// TIA Portal project "Software Day8" (V15)

(* hardware
DEVICE "S7-1200 station_1"  S7-1200 Station
   slot 0: "Rack_0"  S7-1200 Rack  Rack  V1.0
   slot 1: "PLC_1"  CPU 1215C AC/DC/Rly  6ES7 215-1BG40-0XB0  V4.0
*)

// ===== PLC "PLC_1"  CPU 1215C AC/DC/Rly =====

VAR_GLOBAL   // PLC tag table "Default tag table"
   "Tag_1" AT %MD100 : Real;
END_VAR

VAR_GLOBAL   // PLC tag table "VARI"
   "Start" AT %M0.0 : Bool;
   "Pump_A" AT %Q0.0 : Bool;
   "Pump_B" AT %Q0.1 : Bool;
   "Pump_C" AT %Q0.2 : Bool;
   "Mixer Motor" AT %Q0.3 : Bool;
   "Drain Valve" AT %Q0.4 : Bool;
   "Halt" AT %M0.1 : Bool;
   "Empty Sensor" AT %Q0.5 : Bool;
   "Timer 4 CV" AT %MD2 : Time;
   "Stop" AT %M0.2 : Bool;
   "Reset" AT %M0.3 : Bool;
   "Pump A Value" AT %MW64 : Word;
   "Pump B Value" AT %MW66 : Word;
   "Pump C Value" AT %MW68 : Word;
   "Pump A Norm" AT %MD6 : Real;
   "Pump B Norm" AT %MD10 : Real;
   "Pump C Norm" AT %MD14 : Real;
   "Pump A Scaled" AT %MD18 : Real;
   "Pump B Scaled" AT %MD22 : Real;
   "Pump C Scaled" AT %MD26 : Real;
   "Pump A Flow" AT %MD30 : Real;
   "Pump B Flow" AT %MD34 : Real;
   "Pump C Flow" AT %MD38 : Real;
   "Current Level" AT %MD42 : Real;
   "Previous Level" AT %MD46 : Real;
   "Actual Flow Rate" AT %MD50 : Real;
   "ETT" AT %MD54 : DInt;
   "Elapsed Time" AT %MD58 : Real;
   "Expected Flow Rate" AT %MD72 : Real;
   "Flow Rate Diff" AT %MD76 : Real;
   "Flow Rate Mismatch" AT %Q0.7 : Bool;
   "High Level Sensor" AT %Q1.0 : Bool;
   "RED ALARM" AT %Q1.1 : Bool;
   "Current Cycle State" AT %Q1.2 : Bool;
   "Current Step" AT %MW10 : Int;
   "Start Next Cycle" AT %M0.4 : Bool;
   "Flow Rate Difference" AT %MD80 : Real;
END_VAR

// folder: System blocks/Program resources

DATA_BLOCK "IEC_Timer_0_DB"   // DB1
{ S7_Optimized_Access := 'TRUE' }
AUTHOR : Simatic
FAMILY : IEC
NAME : IEC_TMR
VERSION : 1.0
// stored: InstanceOfName IEC_TIMER
"IEC_TIMER"
BEGIN
END_DATA_BLOCK

DATA_BLOCK "IEC_Counter_0_DB"   // DB4
{ S7_Optimized_Access := 'TRUE' }
AUTHOR : Simatic
FAMILY : IEC
NAME : CNTR
VERSION : 1.0
// stored: InstanceOfName IEC_COUNTER
"IEC_COUNTER"
BEGIN
END_DATA_BLOCK

DATA_BLOCK "Timer 1"   // DB6
{ S7_Optimized_Access := 'TRUE' }
AUTHOR : Simatic
FAMILY : IEC
NAME : IEC_TMR
VERSION : 1.0
// stored: InstanceOfName IEC_TIMER
"IEC_TIMER"
BEGIN
END_DATA_BLOCK

DATA_BLOCK "Timer 2"   // DB7
{ S7_Optimized_Access := 'TRUE' }
AUTHOR : Simatic
FAMILY : IEC
NAME : IEC_TMR
VERSION : 1.0
// stored: InstanceOfName IEC_TIMER
"IEC_TIMER"
BEGIN
END_DATA_BLOCK

DATA_BLOCK "Timer 3"   // DB8
{ S7_Optimized_Access := 'TRUE' }
AUTHOR : Simatic
FAMILY : IEC
NAME : IEC_TMR
VERSION : 1.0
// stored: InstanceOfName IEC_TIMER
"IEC_TIMER"
BEGIN
END_DATA_BLOCK

DATA_BLOCK "Timer 4"   // DB9
{ S7_Optimized_Access := 'TRUE' }
AUTHOR : Simatic
FAMILY : IEC
NAME : IEC_TMR
VERSION : 1.0
// stored: InstanceOfName IEC_TIMER
"IEC_TIMER"
BEGIN
END_DATA_BLOCK

// folder: (top level)

ORGANIZATION_BLOCK "Main"   // OB1, LAD, ProgramCycle
TITLE = "Main Program Sweep (Cycle)"
{ S7_Optimized_Access := 'TRUE' }
VERSION : 0.1
// The "Smart" Chemical Dosing Tank (Difficulty: Advanced - Capstone)
// 
// Scenario:
// A tank must mix 3 liquids (A, B, and C) according to a recipe. The PLC controls the pumps using timers. However, the pumps wear out, so the PLC auto-adjusts the timer presets based on a real-time flow rate derived from level sensors.
// 
// 1. Sequential Filling (Timers):
// High_Level (At 90% full).
// Outputs: Pump_A, Pump_B, Pump_C, Mixer_Motor, Drain_Valve.
// Turn on Pump_A for Preset_A seconds. Stop it. Turn on Pump_B for Preset_B seconds. Stop it. Turn on Pump_C for Preset_C seconds. Stop it. Then run the Mixer Motor for 10 seconds. Finally, open the Drain_Valve until the Empty_Sensor triggers. This is a continuous batch cycle.
// 
// 2. Batch Counter (Counters): Use a CTU to count how many complete batches (drain cycles) are finished.
// 
// 3. Adaptive Flow Correction (Math & Comparators):
// Premise: Pump_A is supposed to deliver 100 Liters. The level sensor at 50% represents 500 Liters.
// Read the analog Tank_Level during the fill cycle. Calculate the Actual Flow Rate = (Current_Level - Previous_Level) / Elapsed_Time.
// 
// 4. Use a Comparator. If the Actual Flow Rate is LES than the Expected_Flow_Rate by more than 10%:
// Safety Interlock (Comparators): If the High_Level sensor triggers before Pump_C finishes its timer, immediately stop all pumps and sound a massive alarm.
   VAR_INPUT
      Initial_Call : Bool;   // Initial call of this OB
      Remanence : Bool;   // =True, if remanent data are available
   END_VAR
   VAR_TEMP   // added for the SCL form of the ladder/FBD networks
      _w1 : Bool;
      _w2 : Bool;
   END_VAR
BEGIN

REGION Network 1
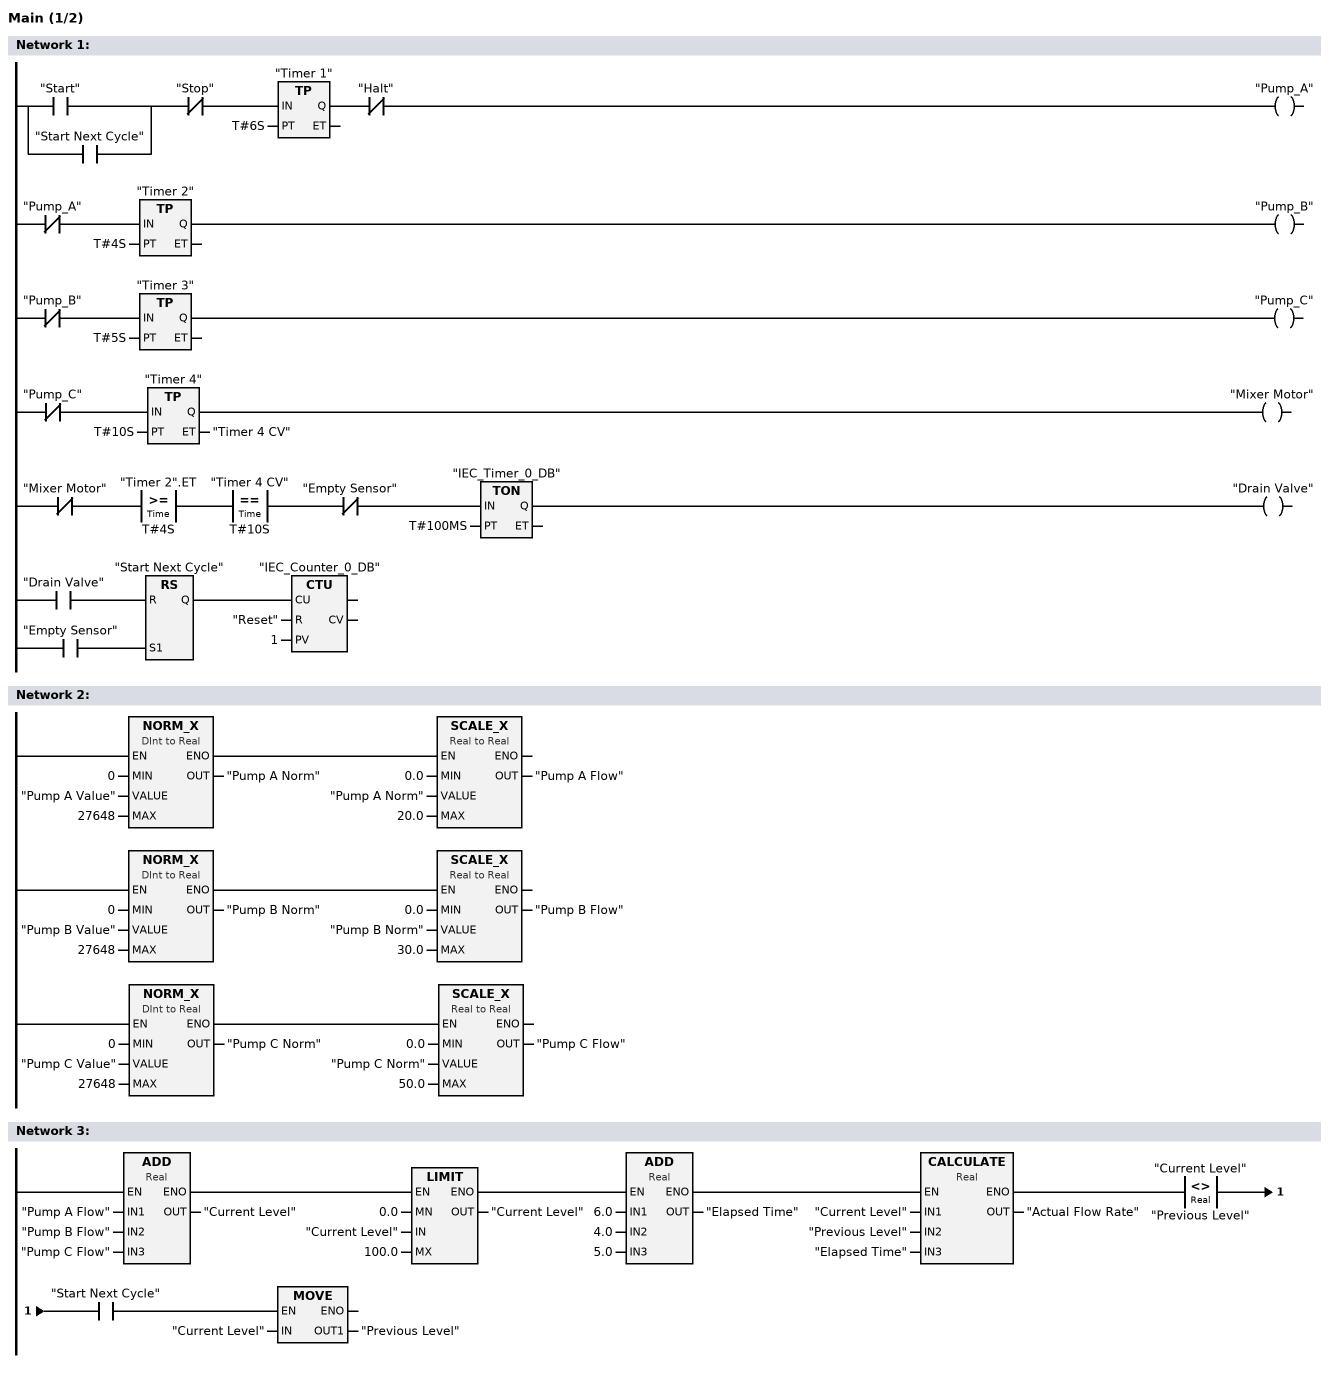
   "Timer 1".TP(IN := ("Start" OR "Start Next Cycle") AND NOT "Stop", PT := T#6S);
   "Pump_A" := "Timer 1".Q AND NOT "Halt";
   "Timer 2".TP(IN := NOT "Pump_A", PT := T#4S);
   "Pump_B" := "Timer 2".Q;
   "Timer 3".TP(IN := NOT "Pump_B", PT := T#5S);
   "Pump_C" := "Timer 3".Q;
   "Timer 4".TP(IN := NOT "Pump_C", PT := T#10S, ET => "Timer 4 CV");
   "Mixer Motor" := "Timer 4".Q;
   "IEC_Timer_0_DB".TON(IN := NOT "Mixer Motor" AND ("Timer 2".ET >= T#4S) AND ("Timer 4 CV" = T#10S) AND NOT "Empty Sensor",
                        PT := T#100MS);
   "Drain Valve" := "IEC_Timer_0_DB".Q;
   IF "Drain Valve" THEN
       "Start Next Cycle" := FALSE;   // RS flip-flop
   END_IF;
   IF "Empty Sensor" THEN "Start Next Cycle" := TRUE; END_IF;
   "IEC_Counter_0_DB".CTU(CU := "Start Next Cycle", R := "Reset", PV := 1);
END_REGION

REGION Network 2
   RUNG wire#powerrail
      { S7_Templates := "[SrcType := DInt, DestType := Real]" } Normalize(min := 0, value := "Pump A Value", max := 27648, out => "Pump A Norm")
      { S7_Templates := "[SrcType := Real, DestType := Real]" } Scale(min := 0.0, value := "Pump A Norm", max := 20.0, out => "Pump A Flow")
   END_RUNG
   RUNG wire#powerrail
      { S7_Templates := "[SrcType := DInt, DestType := Real]" } Normalize(min := 0, value := "Pump B Value", max := 27648, out => "Pump B Norm")
      { S7_Templates := "[SrcType := Real, DestType := Real]" } Scale(min := 0.0, value := "Pump B Norm", max := 30.0, out => "Pump B Flow")
   END_RUNG
   RUNG wire#powerrail
      { S7_Templates := "[SrcType := DInt, DestType := Real]" } Normalize(min := 0, value := "Pump C Value", max := 27648, out => "Pump C Norm")
      { S7_Templates := "[SrcType := Real, DestType := Real]" } Scale(min := 0.0, value := "Pump C Norm", max := 50.0, out => "Pump C Flow")
   END_RUNG
   // the same network as SCL:
   "Pump A Norm" := NORM_X(MIN := 0, VALUE := "Pump A Value", MAX := 27648);
   "Pump A Flow" := SCALE_X(MIN := 0.0, VALUE := "Pump A Norm", MAX := 20.0);
   "Pump B Norm" := NORM_X(MIN := 0, VALUE := "Pump B Value", MAX := 27648);
   "Pump B Flow" := SCALE_X(MIN := 0.0, VALUE := "Pump B Norm", MAX := 30.0);
   "Pump C Norm" := NORM_X(MIN := 0, VALUE := "Pump C Value", MAX := 27648);
   "Pump C Flow" := SCALE_X(MIN := 0.0, VALUE := "Pump C Norm", MAX := 50.0);
END_REGION

REGION Network 3
   "Current Level" := "Pump A Flow" + "Pump B Flow" + "Pump C Flow";
   "Current Level" := LIMIT(MN := 0.0, IN := "Current Level", MX := 100.0);
   "Elapsed Time" := 6.0 + 4.0 + 5.0;
   "Actual Flow Rate" := ("Current Level"-"Previous Level")/("Elapsed Time");
   IF ("Current Level" <> "Previous Level") AND "Start Next Cycle" THEN
       "Previous Level" := "Current Level";
   END_IF;
END_REGION

REGION Network 4
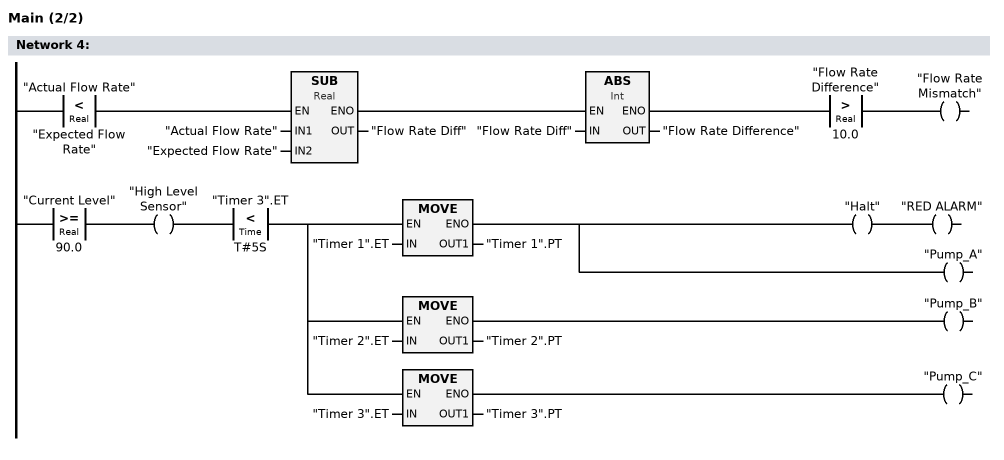
   RUNG wire#powerrail
      { S7_Templates := "SrcType := Real" } LT_Contact(in1 := "Actual Flow Rate", in2 := "Expected Flow Rate")
      { S7_Templates := "SrcType := Real" } Sub(in1 := "Actual Flow Rate", in2 := "Expected Flow Rate", out => "Flow Rate Diff")
      { S7_Templates := "SrcType := Int" } Abs(in := "Flow Rate Diff", out => "Flow Rate Difference")
      { S7_Templates := "SrcType := Real" } GT_Contact(in1 := "Flow Rate Difference", in2 := 10.0)
      Coil( "Flow Rate Mismatch" )
   END_RUNG
   RUNG wire#powerrail
      { S7_Templates := "SrcType := Real" } GE_Contact(in1 := "Current Level", in2 := 90.0)
      Coil( "High Level Sensor" )
      { S7_Templates := "SrcType := Time" } LT_Contact(in1 := "Timer 3".ET, in2 := T#5S)
      wire#w1
      Move(in := "Timer 1".ET, out1 => "Timer 1".PT)
      wire#w2
      Coil( "Halt" )
      Coil( "RED ALARM" )
   END_RUNG
   RUNG wire#w2
      Coil( "Pump_A" )
   END_RUNG
   RUNG wire#w1
      Move(in := "Timer 2".ET, out1 => "Timer 2".PT)
      Coil( "Pump_B" )
   END_RUNG
   RUNG wire#w1
      Move(in := "Timer 3".ET, out1 => "Timer 3".PT)
      Coil( "Pump_C" )
   END_RUNG
   // the same network as SCL:
   #_w1 := "Actual Flow Rate" < "Expected Flow Rate";
   IF #_w1 THEN
       "Flow Rate Diff" := "Actual Flow Rate" - "Expected Flow Rate";
       "Flow Rate Difference" := ABS("Flow Rate Diff");
   END_IF;
   "Flow Rate Mismatch" := #_w1 AND ("Flow Rate Difference" > 10.0);
   "High Level Sensor" := "Current Level" >= 90.0;
   #_w2 := "High Level Sensor" AND ("Timer 3".ET < T#5S);
   IF #_w2 THEN "Timer 1".PT := "Timer 1".ET; END_IF;
   "Halt" := #_w2;
   "RED ALARM" := #_w2;
   "Pump_A" := #_w2;
   IF #_w2 THEN "Timer 2".PT := "Timer 2".ET; END_IF;
   "Pump_B" := #_w2;
   IF #_w2 THEN "Timer 3".PT := "Timer 3".ET; END_IF;
   "Pump_C" := #_w2;
END_REGION
END_ORGANIZATION_BLOCK